PROGRAM PRG_TimestampRegistry
VAR 
	bInit					:BOOL := TRUE;
	fbReadTime				:FB_ReadTime;	
END_VAR

//Init
IF bInit THEN	
	bInit := FALSE;
END_IF

//Call read time
A_ReadTime();
	
//Reset Commands
GVL_HMI.stTimestampCmd.bResetRegistry := FALSE;

ACTION A_ReadTime:
fbReadTime(
	bReset := GVL_HMI.stTimestampCmd.bResetRegistry,
	bSignalIn := GVL_IO.stItemSimulator.bSignalIn,
	aDeltaTimeMS => GVL_HMI.stTimestampStatus.aDeltaTimeMS,
	aDigitalSensorTime => GVL_HMI.stTimestampStatus.aDigitalSensorTime,
	aTCPPortCameraTime => GVL_HMI.stTimestampStatus.aTCPPortCameraTime);
END_ACTION

END_PROGRAM

(* stored: Version 1.1.0.1, ProductVersion 3.1.4024.12
   POU PRG_TimestampRegistry: Id {41809a93-5b53-47f0-b8b5-05c700b2cea3}, SpecialFunc None
   Action A_ReadTime: Id {8e7cafae-cf78-4063-9d90-ae4f1b3eed2e} *)
